TYPE ST_TestStruct :
STRUCT
	by_this	: ST_TestStruct2;
END_STRUCT
END_TYPE

(* stored: Version 1.1.0.1, ProductVersion 3.1.4024.11
   DUT ST_TestStruct: Id {b2fca124-17f1-4244-bd8a-a4255f3df080} *)
